GLOBALCONSTANTS AID_OE (* Output ellipse object attribute ids *)
  (* Standard: 61499-1; Description: Copyright (c) 2023 HR Agrartechnik GmbH This program and the accompanying materials are made available under the terms of the Eclipse Public License 2.0 which is available at https://www.eclipse.org/legal/epl-2.0/ SPDX-License-Identifier: EPL-2.0 *)
  (* Version 1.0, 2026-06-20, Franz Höpfinger, HR Agrartechnik GmbH *)
  PACKAGE isobus::UT::Q::const::AID;
  VAR_GLOBAL CONSTANT
    LINE_ATT : USINT := USINT#1; (* 1: AID_OE_LINE_ATT - Object ID of a Line Attributes object. *)
    WIDTH : USINT := USINT#2; (* 2: AID_OE_WIDTH - Width in pixels. *)
    HEIGHT : USINT := USINT#3; (* 3: AID_OE_HEIGHT - Height in pixels. *)
    ELLIPSE_TYPE : USINT := USINT#4; (* 4: AID_OE_ELLIPSE_TYPE - 0=Closed Ellipse, 1=Open Ellipse, 2=Closed Segment, 3=Closed Section. *)
    START_ANGLE : USINT := USINT#5; (* 5: AID_OE_START_ANGLE *)
    END_ANGLE : USINT := USINT#6; (* 6: AID_OE_END_ANGLE *)
    FILL_ATT : USINT := USINT#7; (* 7: AID_OE_FILL_ATT - Object ID of a Fill Attributes object. *)
  END_VAR
END_GLOBALCONSTANTS
